(* PLC project Tc2_IoFunctions.IOF_SER_SetPhase Demo, tc3-libraries-kb TwinCAT 3.1 *)
(* stored: creationDateTime 2026-05-21T00:00:00, modificationDateTime 2026-05-21T00:00:00 *)

PROGRAM P_Demo_IOF_SER_SetPhase
  VAR
    fbSercosSetPhase : IOF_SER_SetPhase;  (* SERCOS phase 切换 FB *)
    sLocalNetId : T_AmsNetId := '';  (* 本机 *)
    nSercosDeviceId : UDINT := 1;  (* 主站 Device Id *)
    nTargetPhaseValue : BYTE := 2;  (* 目标 phase 值 (0..4) *)
    bSetPhaseReq : BOOL := FALSE;  (* 上升沿触发切换 *)
    tSetPhaseTimeout : TIME := T#15S;  (* 超时（phase 切换较慢） *)
    bSetPhaseBusy : BOOL;  (* 工作中 *)
    bSetPhaseErr : BOOL;  (* 出错 *)
    nLastErrCode : UDINT;  (* 错误号 *)
  END_VAR

// =============================================================================
// 场景：调试期：HMI 按"进入调试模式"按钮 → 把 SERCOS 环切到 phase 2 让参数可访问。
// 价值：让"参数调试"成为正式工序的一部分。
// 验证：**先停所有 motion** → 写 nTargetPhaseValue := 2、bSetPhaseReq := TRUE → bSetPhaseBusy 短暂 TRUE → 回 FALSE 后用 IOF_SER_GetPhase 确认 phase = 2。
// 验证步骤：
//   1. 右键 PLC 项目 → Import PLCopenXML → 选本文件
//   2. 引用 Tc2_IoFunctions（References → Add library）
//   3. 编译 → 登录 → 运行；按上方『验证』行的指示在线写值观察
// =============================================================================

// 警告：从 phase 4 切回低 phase 会停所有 motion；先确保 drive 已 disable
fbSercosSetPhase(
    NETID    := sLocalNetId,
    DEVICEID := nSercosDeviceId,
    PHASE    := nTargetPhaseValue,
    SET      := bSetPhaseReq,
    TMOUT    := tSetPhaseTimeout,
    BUSY     => bSetPhaseBusy,
    ERR      => bSetPhaseErr,
    ERRID    => nLastErrCode
);
END_PROGRAM
